TYPE ST_AxisInputs :
STRUCT
	
///////Axis Inputs///////
	bLimitFwd 	AT %I*	:	BOOL;			//Forward limit switch
	bLimitBwd 	AT %I*	:	BOOL;			//Backward limit switch
	bHomeSensor AT %I*	:	BOOL;			//Reference siganl for homing
	bEncLAtch 	AT %I*	: 	BOOL;			//Reference index signal from inc. enconder
	
END_STRUCT
END_TYPE

(* stored: Version 1.1.0.1, ProductVersion 3.1.4022.12
   DUT ST_AxisInputs: Id {c688a7fd-4b78-4e23-92c9-09a1ce1d0174} *)
